// LS Electric XG5000 project: Tip-off System_230829-1_modbus
// 기종:PLC_K80S 제목: 회사: 저자: 설명: 
// PLC LSPLC
// module base 0 slot 0: 입출력 모듈:XBM-DN/DP32H2 (DC 24V입력/TR 출력, 32점)
// module base 0 slot 1: 내장위치결정:XBF-PO02E (오픈컬렉터형, 2축)
// module base 0 slot 2: 입력 모듈:XBE-DC16A/B (DC24V 입력, 16점 / DC12/24V 입력, 16점)
// module base 0 slot 3: 입력 모듈:XBE-DC16A/B (DC24V 입력, 16점 / DC12/24V 입력, 16점)
// module base 0 slot 4: 출력 모듈:XBE-RY16A (릴레이 출력, 16점 (2A용, 8점/COM))
// module base 0 slot 5: 출력 모듈:XBE-RY16A (릴레이 출력, 16점 (2A용, 8점/COM))

PROGRAM NewProgram (task: 스캔 프로그램)

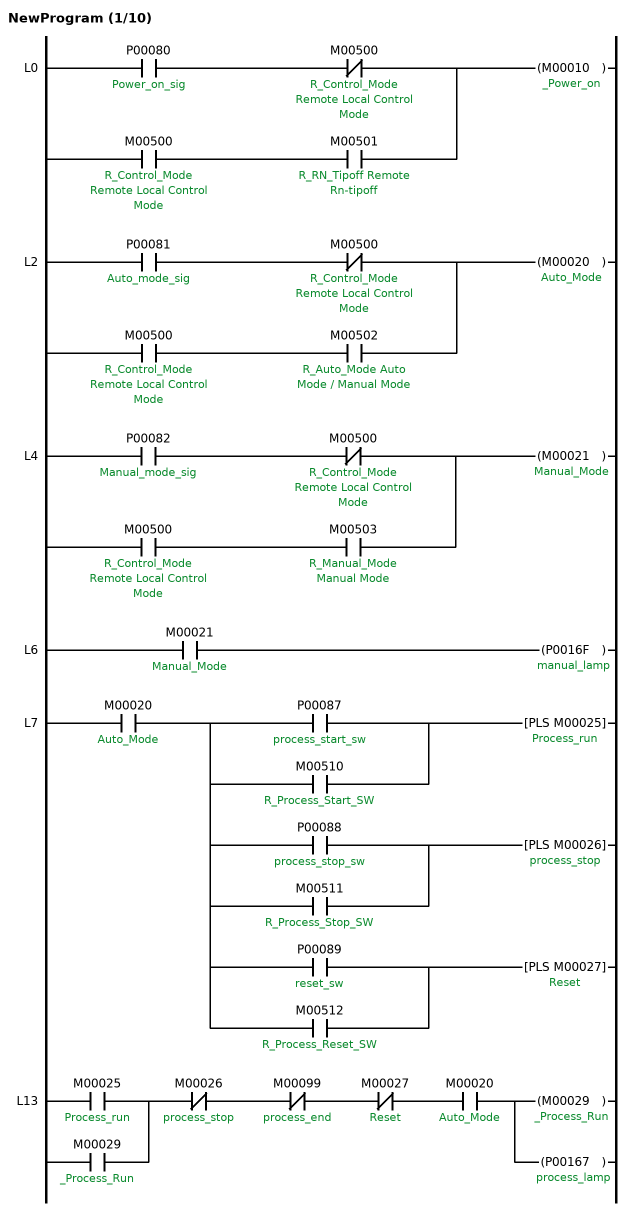
; L0
LOAD      P00080	// Power_on_sig
AND NOT   M00500	// R_Control_Mode Remote Local Control Mode
LOAD      M00500	// R_Control_Mode Remote Local Control Mode
AND       M00501	// R_RN_Tipoff Remote Rn-tipoff
OR LOAD
OUT       M00010	// _Power_on
; L2
LOAD      P00081	// Auto_mode_sig
AND NOT   M00500	// R_Control_Mode Remote Local Control Mode
LOAD      M00500	// R_Control_Mode Remote Local Control Mode
AND       M00502	// R_Auto_Mode Auto Mode / Manual Mode
OR LOAD
OUT       M00020	// Auto_Mode
; L4
LOAD      P00082	// Manual_mode_sig
AND NOT   M00500	// R_Control_Mode Remote Local Control Mode
LOAD      M00500	// R_Control_Mode Remote Local Control Mode
AND       M00503	// R_Manual_Mode Manual Mode
OR LOAD
OUT       M00021	// Manual_Mode
; L6
LOAD      M00021	// Manual_Mode
OUT       P0016F	// manual_lamp
; L7
LOAD      M00020	// Auto_Mode
MPUSH
LOAD      P00087	// process_start_sw
OR        M00510	// R_Process_Start_SW
AND LOAD
OUTP      M00025	// Process_run
MLOAD
LOAD      P00088	// process_stop_sw
OR        M00511	// R_Process_Stop_SW
AND LOAD
OUTP      M00026	// process_stop
MPOP
LOAD      P00089	// reset_sw
OR        M00512	// R_Process_Reset_SW
AND LOAD
OUTP      M00027	// Reset
; L13
LOAD      M00025	// Process_run
OR        M00029	// _Process_Run
AND NOT   M00026	// process_stop
AND NOT   M00099	// process_end
AND NOT   M00027	// Reset
AND       M00020	// Auto_Mode
OUT       M00029	// _Process_Run
OUT       P00167	// process_lamp

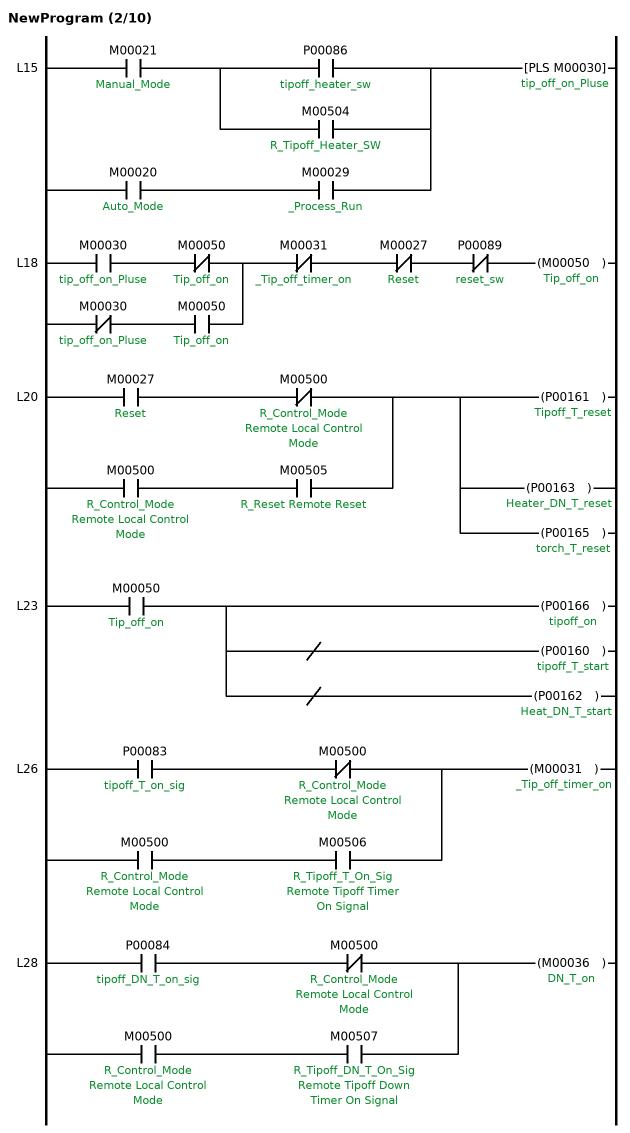
; L15
LOAD      M00021	// Manual_Mode
LOAD      P00086	// tipoff_heater_sw
OR        M00504	// R_Tipoff_Heater_SW
AND LOAD
LOAD      M00020	// Auto_Mode
AND       M00029	// _Process_Run
OR LOAD
OUTP      M00030	// tip_off_on_Pluse
; L18
LOAD      M00030	// tip_off_on_Pluse
AND NOT   M00050	// Tip_off_on
LOAD NOT  M00030	// tip_off_on_Pluse
AND       M00050	// Tip_off_on
OR LOAD
AND NOT   M00031	// _Tip_off_timer_on
AND NOT   M00027	// Reset
AND NOT   P00089	// reset_sw
OUT       M00050	// Tip_off_on
; L20
LOAD      M00027	// Reset
AND NOT   M00500	// R_Control_Mode Remote Local Control Mode
LOAD      M00500	// R_Control_Mode Remote Local Control Mode
AND       M00505	// R_Reset Remote Reset
OR LOAD
OUT       P00161	// Tipoff_T_reset
OUT       P00163	// Heater_DN_T_reset
OUT       P00165	// torch_T_reset
; L23
LOAD      M00050	// Tip_off_on
OUT       P00166	// tipoff_on
MPUSH
NOT
OUT       P00160	// tipoff_T_start
MPOP
NOT
OUT       P00162	// Heat_DN_T_start
; L26
LOAD      P00083	// tipoff_T_on_sig
AND NOT   M00500	// R_Control_Mode Remote Local Control Mode
LOAD      M00500	// R_Control_Mode Remote Local Control Mode
AND       M00506	// R_Tipoff_T_On_Sig Remote Tipoff Timer On Signal
OR LOAD
OUT       M00031	// _Tip_off_timer_on
; L28
LOAD      P00084	// tipoff_DN_T_on_sig
AND NOT   M00500	// R_Control_Mode Remote Local Control Mode
LOAD      M00500	// R_Control_Mode Remote Local Control Mode
AND       M00507	// R_Tipoff_DN_T_On_Sig Remote Tipoff Down Timer On Signal
OR LOAD
OUT       M00036	// DN_T_on

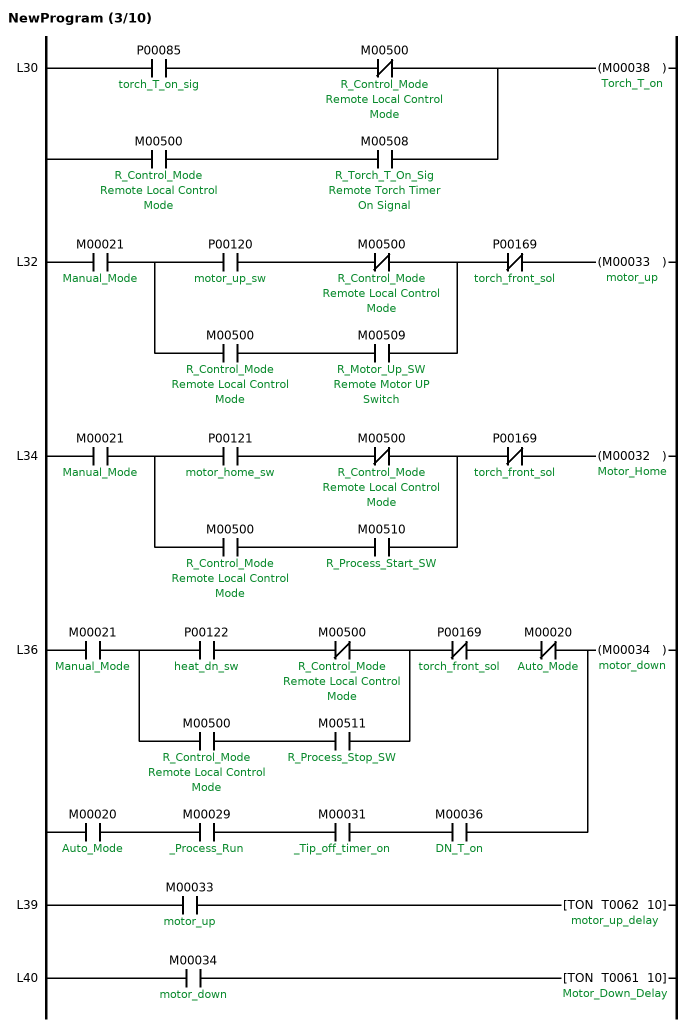
; L30
LOAD      P00085	// torch_T_on_sig
AND NOT   M00500	// R_Control_Mode Remote Local Control Mode
LOAD      M00500	// R_Control_Mode Remote Local Control Mode
AND       M00508	// R_Torch_T_On_Sig Remote Torch Timer On Signal
OR LOAD
OUT       M00038	// Torch_T_on
; L32
LOAD      M00021	// Manual_Mode
LOAD      P00120	// motor_up_sw
AND NOT   M00500	// R_Control_Mode Remote Local Control Mode
LOAD      M00500	// R_Control_Mode Remote Local Control Mode
AND       M00509	// R_Motor_Up_SW Remote Motor UP Switch
OR LOAD
AND LOAD
AND NOT   P00169	// torch_front_sol
OUT       M00033	// motor_up
; L34
LOAD      M00021	// Manual_Mode
LOAD      P00121	// motor_home_sw
AND NOT   M00500	// R_Control_Mode Remote Local Control Mode
LOAD      M00500	// R_Control_Mode Remote Local Control Mode
AND       M00510	// R_Process_Start_SW
OR LOAD
AND LOAD
AND NOT   P00169	// torch_front_sol
OUT       M00032	// Motor_Home
; L36
LOAD      M00021	// Manual_Mode
LOAD      P00122	// heat_dn_sw
AND NOT   M00500	// R_Control_Mode Remote Local Control Mode
LOAD      M00500	// R_Control_Mode Remote Local Control Mode
AND       M00511	// R_Process_Stop_SW
OR LOAD
AND LOAD
AND NOT   P00169	// torch_front_sol
AND NOT   M00020	// Auto_Mode
LOAD      M00020	// Auto_Mode
AND       M00029	// _Process_Run
AND       M00031	// _Tip_off_timer_on
AND       M00036	// DN_T_on
OR LOAD
OUT       M00034	// motor_down
; L39
LOAD      M00033	// motor_up
TON       T0062 10	// motor_up_delay
; L40
LOAD      M00034	// motor_down
TON       T0061 10	// Motor_Down_Delay

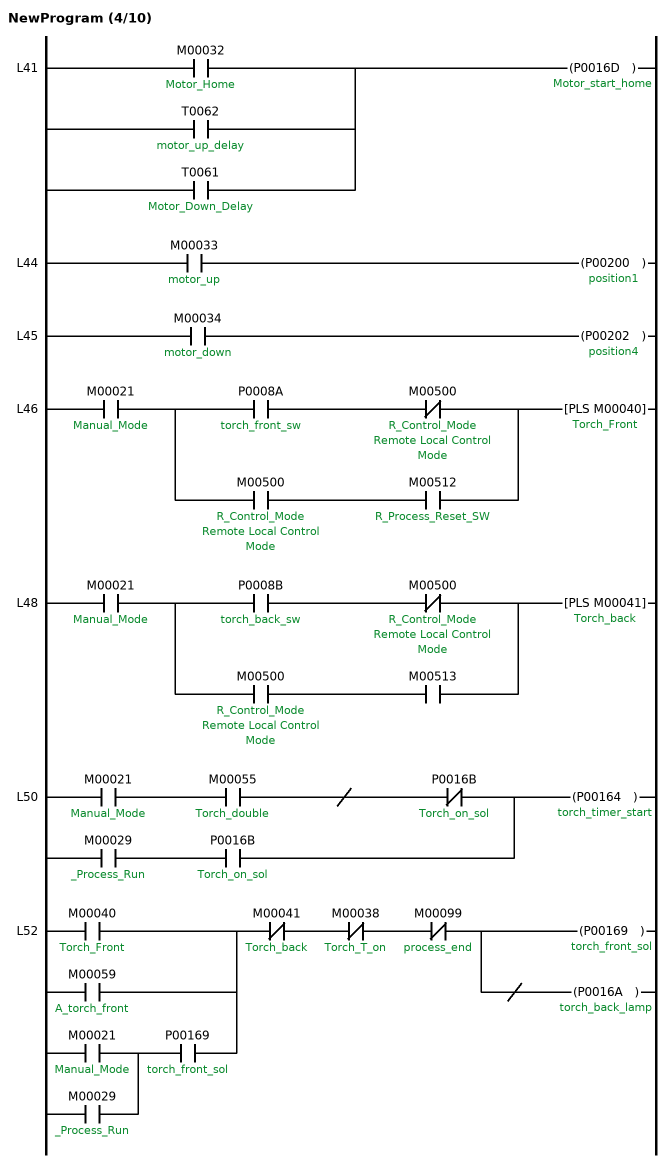
; L41
LOAD      M00032	// Motor_Home
OR        T0062	// motor_up_delay
OR        T0061	// Motor_Down_Delay
OUT       P0016D	// Motor_start_home
; L44
LOAD      M00033	// motor_up
OUT       P00200	// position1
; L45
LOAD      M00034	// motor_down
OUT       P00202	// position4
; L46
LOAD      M00021	// Manual_Mode
LOAD      P0008A	// torch_front_sw
AND NOT   M00500	// R_Control_Mode Remote Local Control Mode
LOAD      M00500	// R_Control_Mode Remote Local Control Mode
AND       M00512	// R_Process_Reset_SW
OR LOAD
AND LOAD
OUTP      M00040	// Torch_Front
; L48
LOAD      M00021	// Manual_Mode
LOAD      P0008B	// torch_back_sw
AND NOT   M00500	// R_Control_Mode Remote Local Control Mode
LOAD      M00500	// R_Control_Mode Remote Local Control Mode
AND       M00513
OR LOAD
AND LOAD
OUTP      M00041	// Torch_back
; L50
LOAD      M00021	// Manual_Mode
AND       M00055	// Torch_double
NOT
AND NOT   P0016B	// Torch_on_sol
LOAD      M00029	// _Process_Run
AND       P0016B	// Torch_on_sol
OR LOAD
OUT       P00164	// torch_timer_start
; L52
LOAD      M00040	// Torch_Front
OR        M00059	// A_torch_front
LOAD      M00021	// Manual_Mode
OR        M00029	// _Process_Run
AND       P00169	// torch_front_sol
OR LOAD
AND NOT   M00041	// Torch_back
AND NOT   M00038	// Torch_T_on
AND NOT   M00099	// process_end
OUT       P00169	// torch_front_sol
NOT
OUT       P0016A	// torch_back_lamp

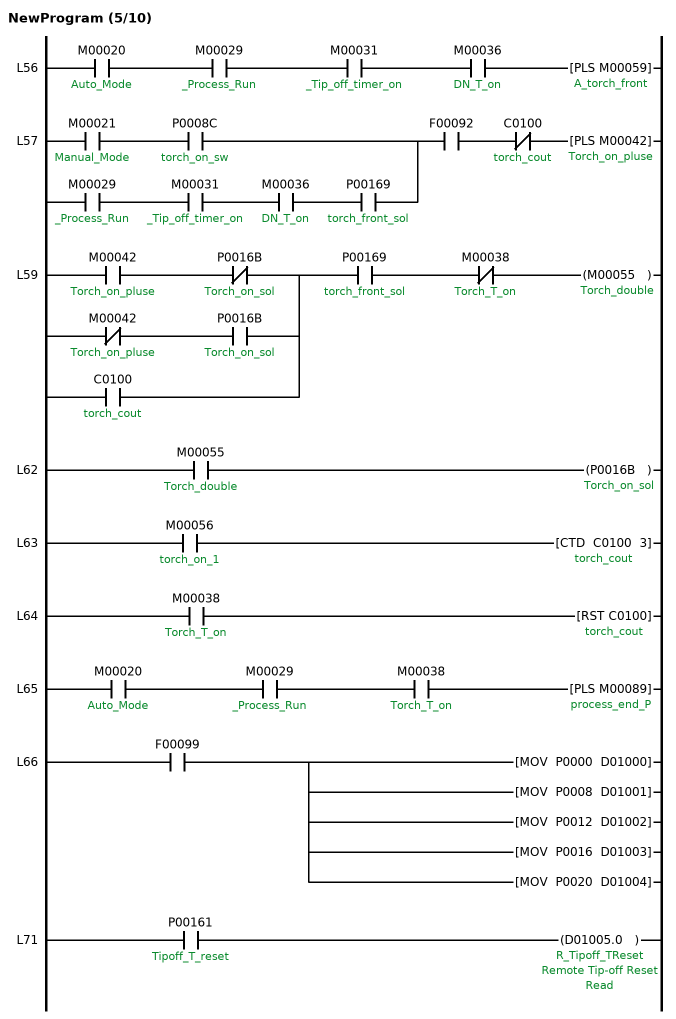
; L56
LOAD      M00020	// Auto_Mode
AND       M00029	// _Process_Run
AND       M00031	// _Tip_off_timer_on
AND       M00036	// DN_T_on
OUTP      M00059	// A_torch_front
; L57
LOAD      M00021	// Manual_Mode
AND       P0008C	// torch_on_sw
LOAD      M00029	// _Process_Run
AND       M00031	// _Tip_off_timer_on
AND       M00036	// DN_T_on
AND       P00169	// torch_front_sol
OR LOAD
AND       F00092
AND NOT   C0100	// torch_cout
OUTP      M00042	// Torch_on_pluse
; L59
LOAD      M00042	// Torch_on_pluse
AND NOT   P0016B	// Torch_on_sol
LOAD NOT  M00042	// Torch_on_pluse
AND       P0016B	// Torch_on_sol
OR LOAD
OR        C0100	// torch_cout
AND       P00169	// torch_front_sol
AND NOT   M00038	// Torch_T_on
OUT       M00055	// Torch_double
; L62
LOAD      M00055	// Torch_double
OUT       P0016B	// Torch_on_sol
; L63
LOAD      M00056	// torch_on_1
CTD       C0100 3	// torch_cout
; L64
LOAD      M00038	// Torch_T_on
RST       C0100	// torch_cout
; L65
LOAD      M00020	// Auto_Mode
AND       M00029	// _Process_Run
AND       M00038	// Torch_T_on
OUTP      M00089	// process_end_P
; L66
LOAD      F00099
MOV       P0000 D01000
MOV       P0008 D01001
MOV       P0012 D01002
MOV       P0016 D01003
MOV       P0020 D01004
; L71
LOAD      P00161	// Tipoff_T_reset
OUT       D01005.0	// R_Tipoff_TReset Remote Tip-off Reset Read

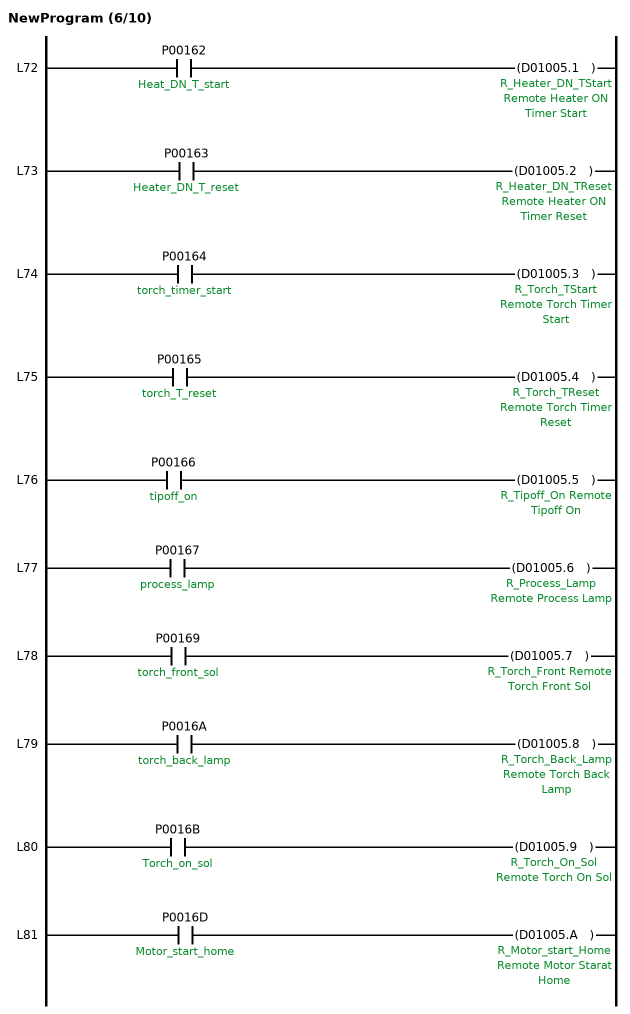
; L72
LOAD      P00162	// Heat_DN_T_start
OUT       D01005.1	// R_Heater_DN_TStart Remote Heater ON Timer Start
; L73
LOAD      P00163	// Heater_DN_T_reset
OUT       D01005.2	// R_Heater_DN_TReset Remote Heater ON Timer Reset
; L74
LOAD      P00164	// torch_timer_start
OUT       D01005.3	// R_Torch_TStart Remote Torch Timer Start
; L75
LOAD      P00165	// torch_T_reset
OUT       D01005.4	// R_Torch_TReset Remote Torch Timer Reset
; L76
LOAD      P00166	// tipoff_on
OUT       D01005.5	// R_Tipoff_On Remote Tipoff On
; L77
LOAD      P00167	// process_lamp
OUT       D01005.6	// R_Process_Lamp Remote Process Lamp
; L78
LOAD      P00169	// torch_front_sol
OUT       D01005.7	// R_Torch_Front Remote Torch Front Sol
; L79
LOAD      P0016A	// torch_back_lamp
OUT       D01005.8	// R_Torch_Back_Lamp Remote Torch Back Lamp
; L80
LOAD      P0016B	// Torch_on_sol
OUT       D01005.9	// R_Torch_On_Sol Remote Torch On Sol
; L81
LOAD      P0016D	// Motor_start_home
OUT       D01005.A	// R_Motor_start_Home Remote Motor Starat Home

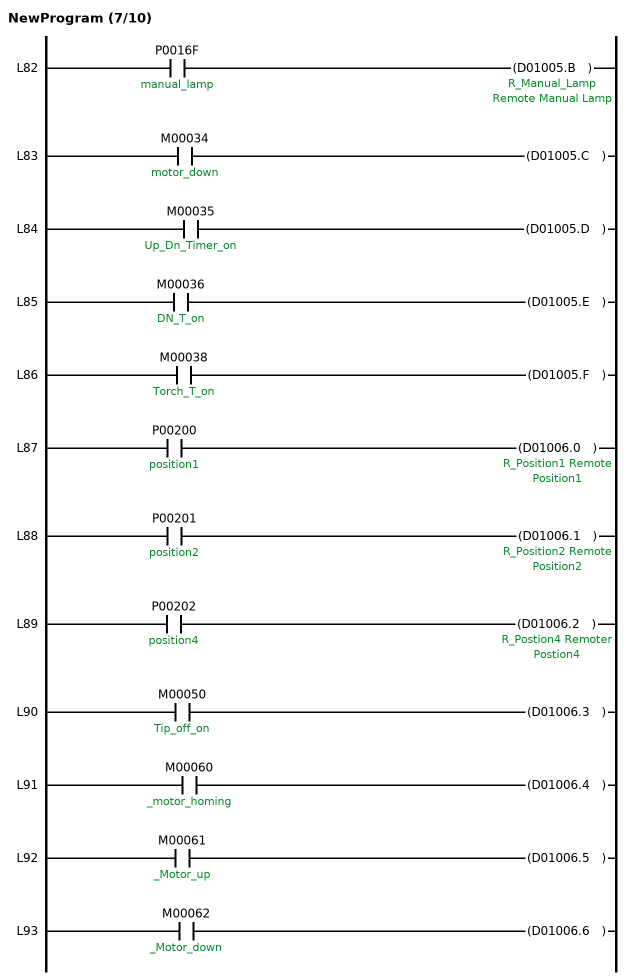
; L82
LOAD      P0016F	// manual_lamp
OUT       D01005.B	// R_Manual_Lamp Remote Manual Lamp
; L83
LOAD      M00034	// motor_down
OUT       D01005.C
; L84
LOAD      M00035	// Up_Dn_Timer_on
OUT       D01005.D
; L85
LOAD      M00036	// DN_T_on
OUT       D01005.E
; L86
LOAD      M00038	// Torch_T_on
OUT       D01005.F
; L87
LOAD      P00200	// position1
OUT       D01006.0	// R_Position1 Remote Position1
; L88
LOAD      P00201	// position2
OUT       D01006.1	// R_Position2 Remote Position2
; L89
LOAD      P00202	// position4
OUT       D01006.2	// R_Postion4 Remoter Postion4
; L90
LOAD      M00050	// Tip_off_on
OUT       D01006.3
; L91
LOAD      M00060	// _motor_homing
OUT       D01006.4
; L92
LOAD      M00061	// _Motor_up
OUT       D01006.5
; L93
LOAD      M00062	// _Motor_down
OUT       D01006.6

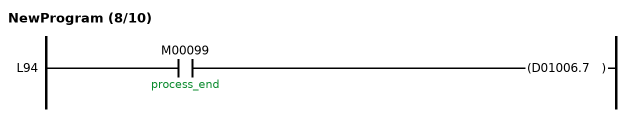
; L94
LOAD      M00099	// process_end
OUT       D01006.7

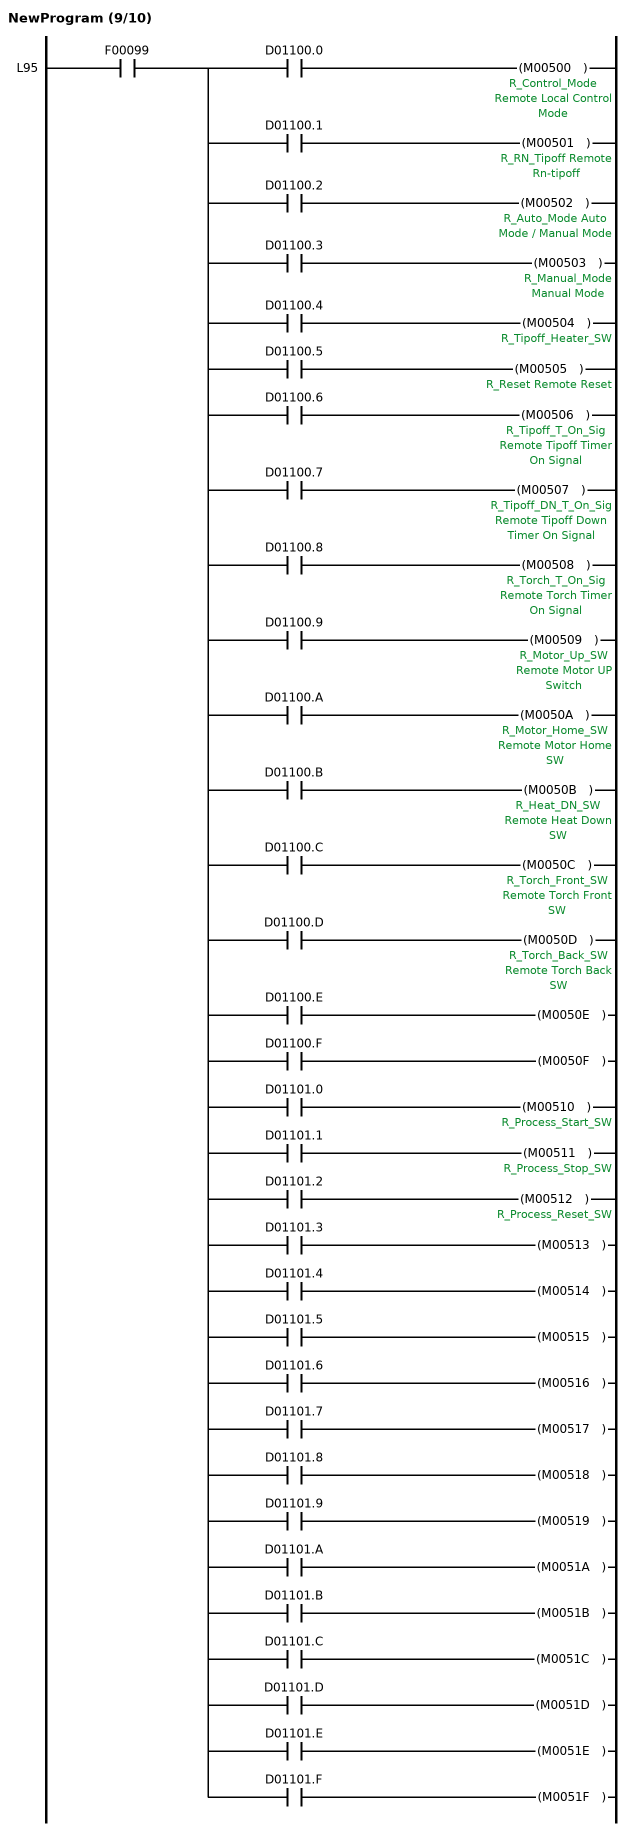
; L95
LOAD      F00099
MPUSH
AND       D01100.0
OUT       M00500	// R_Control_Mode Remote Local Control Mode
MLOAD
AND       D01100.1
OUT       M00501	// R_RN_Tipoff Remote Rn-tipoff
MLOAD
AND       D01100.2
OUT       M00502	// R_Auto_Mode Auto Mode / Manual Mode
MLOAD
AND       D01100.3
OUT       M00503	// R_Manual_Mode Manual Mode
MLOAD
AND       D01100.4
OUT       M00504	// R_Tipoff_Heater_SW
MLOAD
AND       D01100.5
OUT       M00505	// R_Reset Remote Reset
MLOAD
AND       D01100.6
OUT       M00506	// R_Tipoff_T_On_Sig Remote Tipoff Timer On Signal
MLOAD
AND       D01100.7
OUT       M00507	// R_Tipoff_DN_T_On_Sig Remote Tipoff Down Timer On Signal
MLOAD
AND       D01100.8
OUT       M00508	// R_Torch_T_On_Sig Remote Torch Timer On Signal
MLOAD
AND       D01100.9
OUT       M00509	// R_Motor_Up_SW Remote Motor UP Switch
MLOAD
AND       D01100.A
OUT       M0050A	// R_Motor_Home_SW Remote Motor Home SW
MLOAD
AND       D01100.B
OUT       M0050B	// R_Heat_DN_SW Remote Heat Down SW
MLOAD
AND       D01100.C
OUT       M0050C	// R_Torch_Front_SW Remote Torch Front SW
MLOAD
AND       D01100.D
OUT       M0050D	// R_Torch_Back_SW Remote Torch Back SW
MLOAD
AND       D01100.E
OUT       M0050E
MLOAD
AND       D01100.F
OUT       M0050F
MLOAD
AND       D01101.0
OUT       M00510	// R_Process_Start_SW
MLOAD
AND       D01101.1
OUT       M00511	// R_Process_Stop_SW
MLOAD
AND       D01101.2
OUT       M00512	// R_Process_Reset_SW
MLOAD
AND       D01101.3
OUT       M00513
MLOAD
AND       D01101.4
OUT       M00514
MLOAD
AND       D01101.5
OUT       M00515
MLOAD
AND       D01101.6
OUT       M00516
MLOAD
AND       D01101.7
OUT       M00517
MLOAD
AND       D01101.8
OUT       M00518
MLOAD
AND       D01101.9
OUT       M00519
MLOAD
AND       D01101.A
OUT       M0051A
MLOAD
AND       D01101.B
OUT       M0051B
MLOAD
AND       D01101.C
OUT       M0051C
MLOAD
AND       D01101.D
OUT       M0051D
MLOAD
AND       D01101.E
OUT       M0051E
MPOP
AND       D01101.F
OUT       M0051F

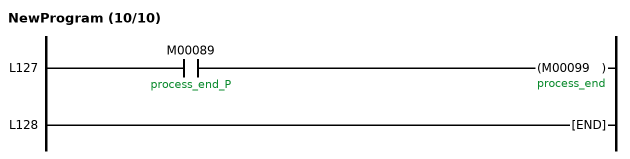
; L127
LOAD      M00089	// process_end_P
OUT       M00099	// process_end
; L128
END

VARIABLES AND COMMENTS (devices not used above)
M00101	BIT	H_L_end
P00100	BIT	H_L_완료
M00105	BIT	H_R_end
T0101	BIT/WORD	H_R_start
M00103	BIT	L_H_end
T0100	BIT/WORD	L_H_start
M00067	BIT	Motor_DN_END
T0060	BIT/WORD	motor_homing_delay
P00055	BIT	motor_out_3
M00063	BIT	Motor_Run_DN_
M00064	BIT	Motor_run_up_
S00201	BIT	motor_step1_up_
S00202	BIT	motor_step2_dn_
S00203	BIT	motor_step3_up_
S00204	BIT	motor_step4_dn_
M00076	BIT	Motor_Strat
M00028	BIT	Process_hold
T0081	BIT/WORD	step1_end
T0080	BIT/WORD	step1_start
T0083	BIT/WORD	step2_end
T0082	BIT/WORD	step2_start
T0085	BIT/WORD	step3_end
T0084	BIT/WORD	step3_start
T0087	BIT/WORD	step4_end
T0086	BIT/WORD	step4_start
M00080	BIT	step_start
T0070	BIT/WORD	tilie_H_L_end
M00071	BIT	tilite_Home
M00100	BIT	Tilite_H_L
M00070	BIT	tilite_L
M00102	BIT	Tilite_L_H
P0004D	BIT	Tilit_Home_sol
S00105	BIT	tilte_1_cycle
C0010	BIT/WORD	tilte_2_cycle
M00073	BIT	tilte_count
T0075	BIT/WORD	Tilte_end
P0000E	BIT	tilte_home_sw
S00101	BIT	Tilte_H_L
M00104	BIT	Tilte_H_R
T0072	BIT/WORD	tilte_H_R_end
P0000D	BIT	tilte_Left_sw
S00102	BIT	Tilte_L_H
T0071	BIT/WORD	Tilte_L_H_end
P0004C	BIT	Tilte_L_sol
S00100	BIT	Tilte_reset
M00072	BIT	tilte_right
P0004E	BIT	tilte_right_sol
P0000F	BIT	tilte_right_sw
S00104	BIT	Tilte_R_H
T0073	BIT/WORD	Tilte_R_H_end
M00085	BIT	torch_start
T0090	BIT/WORD	_torch_front
M00090	BIT	_Torch_start
M00066	BIT	__Motor_Down